// TIA Portal V20 export
DATA_BLOCK "Simulation_DB"   // DB80
// stored: InstanceOfName Unit1.Em2.Simulation, InstanceOfType FB, Namespace Unit1.Em2
"Unit1.Em2.Simulation"
   // VAR
   //    Simulation_addon_Instance { S7_SetPoint := 'True'} : "Simulation_addon";
   //    Simulation_addon_Instance_1 { S7_SetPoint := 'True'} : "Simulation_addon";
   //    Simulation_addon_Instance_2 { S7_SetPoint := 'True'} : "Simulation_addon";
   //    Simulation_addon_Instance_3 { S7_SetPoint := 'True'} : "Simulation_addon";
   //    Simulation_addon_Instance_4 { S7_SetPoint := 'True'} : "Simulation_addon";
   //    Simulation_addon_Instance_5 { S7_SetPoint := 'True'} : "Simulation_addon";
   //    Simulation_addon_Instance_6 { S7_SetPoint := 'True'} : "Simulation_addon";
   //    Simulation_addon_Instance_7 { S7_SetPoint := 'True'} : "Simulation_addon";
   //    Simulation_addon_Instance_8 { S7_SetPoint := 'True'} : "Simulation_addon";
   //    Simulation_addon_Instance_9 { S7_SetPoint := 'True'} : "Simulation_addon";
   //    Simulation_addon_Instance_10 { S7_SetPoint := 'True'} : "Simulation_addon";
   //    Simulation_addon_Instance_11 { S7_SetPoint := 'True'} : "Simulation_addon";
   //    Simulation_addon_Instance_12 { S7_SetPoint := 'True'} : "Simulation_addon";
   //    Simulation_addon_Instance_13 { S7_SetPoint := 'True'} : "Simulation_addon";
   //    Simulation_addon_Instance_14 { S7_SetPoint := 'True'} : "Simulation_addon";
   //    Simulation_addon_Instance_15 { S7_SetPoint := 'True'} : "Simulation_addon";
   //    Simulation_addon_Instance_16 { S7_SetPoint := 'True'} : "Simulation_addon";
   //    Simulation_addon_Instance_17 { S7_SetPoint := 'True'} : "Simulation_addon";
   //    Simulation_addon_Instance_18 { S7_SetPoint := 'True'} : "Simulation_addon";
   //    Simulation_addon_Instance_19 { S7_SetPoint := 'True'} : "Simulation_addon";
   //    Simulation_addon_Instance_20 { S7_SetPoint := 'True'} : "Simulation_addon";
   //    Simulation_addon_Instance_21 { S7_SetPoint := 'True'} : "Simulation_addon";
   // END_VAR
BEGIN
END_DATA_BLOCK
